FUNCTION_BLOCK Contactor
VAR
	_output : BOOL;
END_VAR

PROPERTY State : BOOL
GET
State := _output;
END_GET
SET
_output := State;
END_SET
END_PROPERTY

END_FUNCTION_BLOCK

(* stored: Version 1.1.0.1, ProductVersion 3.1.4024.12
   POU Contactor: Id {c060f755-e854-44d6-80a6-8e4dedcc8084}, SpecialFunc None
   Property State: Id {0e142a4b-cd3f-4ab7-9ab4-1784c7145a1f}
   Get Get: Id {a3074313-4226-4222-a590-1d86a6eb0a5e}
   Set Set: Id {04cd2443-c326-4ff6-9a1d-095275924f65} *)
